// TwinCAT 3 PLC project ICBxx
// Title: ICBxx
// Company: iMusic AS
// Author: Jakob Bak
// ProjectVersion: 0.0.1.0
// Description: TwinCAT Library for ICB* series Inductive Sensors from Carlo Gavazzi
// ProgramVersion: 3.1.4024.0
// libraries:
//   Tc2_Standard, * (Beckhoff Automation GmbH)
//   Tc2_System, * (Beckhoff Automation GmbH)
//   Tc3_Module, * (Beckhoff Automation GmbH)
// project tree:
//   DUTs/ ST_ICBxx.TcDUT
//   / PlcTask.TcTTO
//   POUs/ MAIN.TcPOU
//   Version/ Global_Version.TcGVL
// real-time tasks:
//   TASK PlcTask: cycle T#10ms, priority 20, ADS port 350

CONFIGURATION ICBxx
    RESOURCE PLC ON TwinCAT3
        TASK PlcTask(INTERVAL := T#10ms, PRIORITY := 20);
        PROGRAM MAIN WITH PlcTask : MAIN;
    END_RESOURCE
END_CONFIGURATION

// ---- DUTs/ST_ICBxx.TcDUT
TYPE ST_ICBxx :
STRUCT
	bPresenceDetection 	AT%I* : BIT;
	bFrequencyDetection AT%I* : BIT;
	bTemperatureAlarm	AT%I* : BIT;
	bSwitchingOutput	AT%I* : BIT;
END_STRUCT
END_TYPE

// ---- Version/Global_Version.TcGVL
{attribute 'TcGenerated'}
{attribute 'no-analysis'}
{attribute 'linkalways'}
// This function has been automatically generated from the project information.
VAR_GLOBAL CONSTANT
	{attribute 'const_non_replaced'}
	stLibVersion_ICBxx : ST_LibVersion := (iMajor := 0, iMinor := 0, iBuild := 1, iRevision := 0, nFlags := 0, sVersion := '0.0.1.0');
END_VAR

// ---- POUs/MAIN.TcPOU
PROGRAM MAIN
VAR
END_VAR

END_PROGRAM
